PROGRAM PRG_PMPS
VAR
    fbArbiterIO: FB_SubSysToArbiter_IO;
END_VAR

GVL.fbFastFaultOutput1.Execute(i_xVeto := PMPS_GVL.stCurrentBeamParameters.aVetoDevices[PMPS.L_Stopper.ST1L1]);
fbArbiterIO(
    i_bVeto := PMPS_GVL.stCurrentBeamParameters.aVetoDevices[PMPS.L_Stopper.ST1L1],
    Arbiter:=GVL.fbArbiter1,
    fbFFHWO:=GVL.fbFastFaultOutput1);

END_PROGRAM

(* stored: Version 1.1.0.1, ProductVersion 3.1.4024.6
   POU PRG_PMPS: Id {dff18baf-d3c9-4cb4-be04-4a60c54f1a90}, SpecialFunc None *)
